// An interface for a fully functioning TCPIP control with only method calling
INTERFACE I_TcpIpCommControl

// Connets to the target client with the provided Ip address and port
METHOD Connect : BOOL
VAR_INPUT
	Ipv4Address	: Tc2_System.T_IPv4Addr;	// Ip Address
	Port		: UINT;	// Port
END_VAR
END_METHOD

// Disconnects from the server and closes all active socket connections. Returns TRUE when done.
METHOD Disconnect : BOOL
END_METHOD

{attribute 'monitoring' := 'call'}
PROPERTY Error : BOOL
GET
END_GET
END_PROPERTY

{attribute 'monitoring' := 'call'}
PROPERTY PUBLIC IsConnected : BOOL
GET
END_GET
END_PROPERTY

// Awaits a response from the client and returns TRUE when done. Response string can be found in the refResponse
// Method needs to be called untill TRUE is returned to finish the sending sequence!
METHOD Receive : BOOL
VAR_INPUT
	refResponse	: REFERENCE TO Tc2_System.T_MaxString;	// Response will be written to the string variable here
END_VAR
END_METHOD

{attribute 'monitoring' := 'call'}
(* Gets or sets the reconnect period. 
The value should not be set too low, since timeout periods of > 30 s may occur in the event of a network interruption. 
If the value is too low, command execution would be interrupted prematurely, and ADS error code 1861 (timeout elapsed) 
would be returned instead of the Winsocket error WSAETIMEDOUT.*)
PROPERTY PUBLIC ReconnectPeriod : TIME
GET
END_GET
SET
END_SET
END_PROPERTY

// Sends the command to the client and returns TRUE when done. 
// Method needs to be called untill TRUE is returned to finish the sending sequence!
METHOD Send : BOOL
VAR_INPUT
	sCommand	: Tc2_System.T_MaxString;	// Command to be send
END_VAR
END_METHOD

END_INTERFACE

(* stored: Version 1.1.0.1, ProductVersion 3.1.4024.15
   Itf I_TcpIpCommControl: Id {67043732-a237-03d9-32d4-f101b9201dbd}
   Method Connect: Id {48628900-6f9d-06e4-30d6-4f2ef800c3e2}
   Method Disconnect: Id {b1fe599a-dae1-03f1-3dde-cbee642b75c9}
   Property Error: Id {e988c6ef-45ab-0af2-13a2-77c58972fea1}
   Get Get: Id {93b52573-9911-0715-189c-271862bab6e4}
   Property IsConnected: Id {d9d4ad06-0b47-04e8-2300-5362c4552cd5}
   Get Get: Id {984d42ad-10f9-0fc3-3507-7dba08149b32}
   Method Receive: Id {ba862019-9919-0016-16e9-b800d75a384e}
   Property ReconnectPeriod: Id {d5710ec5-0983-0d82-38f0-54fdb03edc04}
   Get Get: Id {daa213cb-5110-0495-1e33-d0dfe2382bf5}
   Set Set: Id {84f8de42-a6fb-0e3b-2929-5c0a52e7867f}
   Method Send: Id {a058ff05-c22b-08fc-3ab9-c212bd27de3f} *)
